// TIA Portal V17 export
// export: Created 2024-08-26T21:07:22.6616893Z, ExportSetting WithDefaults, DisplayName Totally Integrated Automation Portal, DisplayVersion V17 Update 7, DisplayName TIA Portal Openness, DisplayVersion V17 Update 7, DisplayName TIA Portal Version Control Interface, DisplayVersion V17, DisplayName SINAMICS Startdrive Advanced, DisplayVersion V17 SP2, DisplayName SINAMICS Startdrive G110M, G120, G120C, G120D, G120P, G115D, DisplayVersion V17 SP2, DisplayName SINAMICS Startdrive G130, G150, S120, S150, SINAMICS MV, S210, DisplayVersion V17 SP2, DisplayName STEP 7 Professional, DisplayVersion V17 Update 7, DisplayName STEP 7 Safety, DisplayVersion V17 Update 6, DisplayName WinCC Advanced / Unified PC, DisplayVersion V17 Update 7
TYPE "UDT_Readings"
// stored: IsFailsafeCompliant false
   STRUCT
      Enable : Bool;   // Reading active
      ReaderNumber : USInt;   // Fix (1 to 5) or Manual (10)
      "Name" : String[30];   // Name of Label to read
      LabelType : USInt;   // Master NFP, 2nd NFP, Component Label, batch label
      ReferenceToFound : String[30];   // Reference to be found
      ReferenceStartPosition : USInt;   // Position of reference to be found
      ReferenceLenght : USInt;   // Reference Lenght
      MasterReadingNumber : USInt;   // Reading number of master NFP
      LinkedMasterNumber : USInt;   // Linked number to master NFP
      Message : Array[1.."NumberOfmessages"] of "UDT_IJCoreMessage";   // IJCore Message
   END_STRUCT;
END_TYPE
